# EPICS substitutions: test/simulatorApp/Db/sim_1024.substitutions
file "sim_0256.db" {
pattern { R }
{ "\$(R)0" }
{ "\$(R)1" }
{ "\$(R)2" }
{ "\$(R)3" }
}
